// TIA Portal V18 export
FUNCTION_BLOCK "tp_peter"   // FB40, LAD
{ S7_Optimized_Access := 'TRUE' }
VERSION : 0.1
// stored: AutoNumber true, IsIECCheckEnabled false, IsRetainMemResEnabled false, MemoryReserve 100, SetENOAutomatically false, UDAEnableTagReadback false
   VAR_INPUT
      CLK : Bool;
      pt : Time := T#100ms;
   END_VAR
   VAR_OUTPUT
      Q : Bool;
   END_VAR
   VAR
      was : Bool;
      ton { S7_SetPoint := 'True'} : TON_TIME;
   END_VAR
BEGIN

REGION Network 1
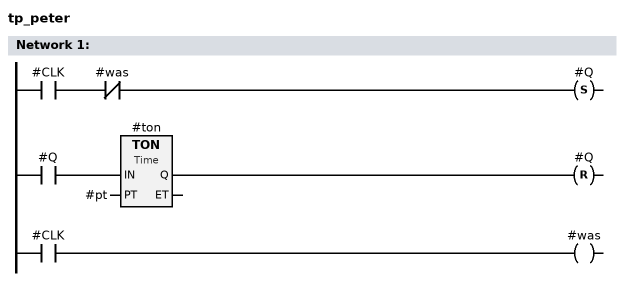
   RUNG wire#powerrail
      Contact( #CLK )
      I_Contact( #was )
      S_Coil( #Q )
   END_RUNG
   RUNG wire#powerrail
      Contact( #Q )
      { S7_Templates := "time_type := Time" } #ton.TON(pt := #pt, et =>)
      R_Coil( #Q )
   END_RUNG
   RUNG wire#powerrail
      Contact( #CLK )
      Coil( #was )
   END_RUNG
   // the same network as SCL:
   IF #CLK AND NOT #was THEN #Q := TRUE; END_IF;
   #ton(IN := #Q, PT := #pt);   // TON
   IF #ton.Q THEN #Q := FALSE; END_IF;
   #was := #CLK;
END_REGION
END_FUNCTION_BLOCK
